PROGRAM MAIN
VAR
	fbRTC : FB_RTCVision;
	
	bFirstCycle: BOOL:= TRUE;
	bInit: BOOL;
	bGetImage: BOOL;
END_VAR

IF bFirstCycle THEN
	bFirstCycle := FALSE;
	
	fbRTC.MR_FirstCycle(	sCameraName := 'RTC 1',
							sClientAmsNetID := '',
							sClientHost := '10.20.254.8',
							tTimeout:=DEFAULT_ADS_TIMEOUT,
							iClientPort := 23);
	bInit := TRUE;
END_IF
if bInit then
	fbRTC.MR_Init();
	
	IF NOT fbRTC.Busy THEN
		bInit := FALSE;
	END_IF
END_IF

if bGetImage then
	fbRTC.MR_GetImage(uStationNumber:=1);
	IF NOT fbRTC.Busy THEN
		bGetImage := false;
	END_IF
END_IF

fbRTC();

END_PROGRAM

(* stored: Version 1.1.0.1, ProductVersion 3.1.4024.9
   POU MAIN: Id {a153987a-a3a6-4662-91fe-3392a52f94e0}, SpecialFunc None *)
